(* Logix 5000 project; controller AB_DataAcquisition 1769-L16ER-BB1B rev 32.11; software revision 32.02 *)

TASK MainTask (continuous, watchdog 500 ms) : MainProgram

MODULES
   Local : 1769-L16ER-BB1B (PointIO 0, rev 32.11)
      Discrete_IO : Embedded (PointIO 1, rev 32.11, Output RPI 20 ms)
END_MODULES

PROGRAM MainProgram   (* main routine MainRoutine *)

ROUTINE MainRoutine   (* ladder *)
END_ROUTINE
END_PROGRAM
